// TIA Portal project "Tuan5" (V16)

(* hardware
DEVICE "S7-1200 station_1"  S7-1200 Station
   slot 0: "Rack_0"  S7-1200 Rack  Rack  V1.0
   slot 1: "PLC_1"  CPU 1214C AC/DC/Rly  6ES7 214-1BG40-0XB0  V4.2
*)

// ===== PLC "PLC_1"  CPU 1214C AC/DC/Rly =====

VAR_GLOBAL   // PLC tag table "Default tag table"
   "Stop" AT %I1.2 : Bool;
   "Quay_thuan" AT %Q0.6 : Bool;
   "Quay_nguoc" AT %Q0.7 : Bool;
   "Start" AT %I1.1 : Bool;
   "Tag_5" AT %I0.1 : Bool;
   "Tag_6" AT %M0.0 : Bool;
   "Tag_7" AT %M0.1 : Bool;
   "Time" AT %MD0 : DWord;
   "Tag_8" AT %M0.3 : Bool;
   "Tag_1" AT %M0.2 : Bool;
   "Tag_2" AT %M2.0 : Bool;
   "Tag_3" AT %Q8.1 : Bool;
   "Tag_4" AT %M0.5 : Bool;
   "Tag_9" AT %M0.4 : Bool;
END_VAR

// folder: System blocks/Program resources

DATA_BLOCK "T1"   // DB1
{ S7_Optimized_Access := 'TRUE' }
AUTHOR : Simatic
FAMILY : IEC
NAME : IEC_TMR
VERSION : 1.0
// stored: InstanceOfName IEC_TIMER
"IEC_TIMER"
BEGIN
END_DATA_BLOCK

DATA_BLOCK "T2"   // DB2
{ S7_Optimized_Access := 'TRUE' }
AUTHOR : Simatic
FAMILY : IEC
NAME : IEC_TMR
VERSION : 1.0
// stored: InstanceOfName IEC_TIMER
"IEC_TIMER"
BEGIN
END_DATA_BLOCK

// folder: (top level)

ORGANIZATION_BLOCK "Main"   // OB1, LAD, ProgramCycle
TITLE = "Main Program Sweep (Cycle)"
{ S7_Optimized_Access := 'TRUE' }
VERSION : 0.1
   VAR_INPUT
      Initial_Call : Bool;   // Initial call of this OB
      Remanence : Bool;   // =True, if remanent data are available
   END_VAR
BEGIN

REGION Network 1
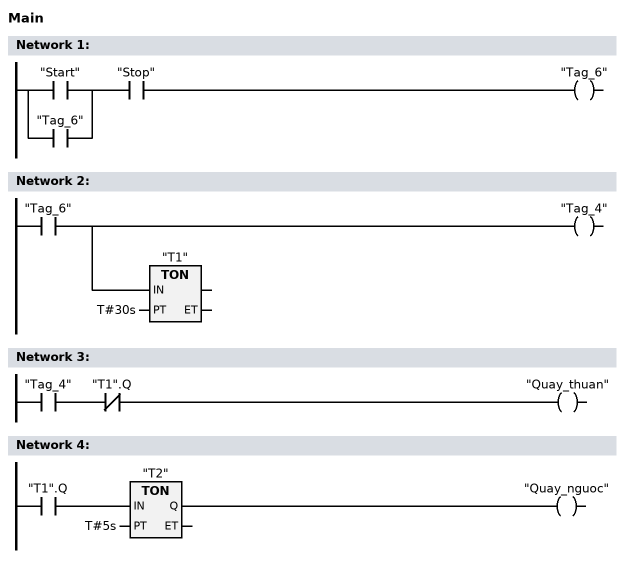
   RUNG wire#powerrail
      Contact( "Start" )
      wire#w1
      Contact( "Stop" )
      Coil( "Tag_6" )
   END_RUNG
   RUNG wire#powerrail
      Contact( "Tag_6" )
   END_RUNG wire#w1
   // the same network as SCL:
   "Tag_6" := ("Start" OR "Tag_6") AND "Stop";
END_REGION

REGION Network 2
   "Tag_4" := "Tag_6";
   "T1".TON(IN := "Tag_6", PT := T#30s);
END_REGION

REGION Network 3
   RUNG wire#powerrail
      Contact( "Tag_4" )
      I_Contact( "T1".Q )
      Coil( "Quay_thuan" )
   END_RUNG
   // the same network as SCL:
   "Quay_thuan" := "Tag_4" AND NOT "T1".Q;
END_REGION

REGION Network 4
   "T2".TON(IN := "T1".Q, PT := T#5s);
   "Quay_nguoc" := "T2".Q;
END_REGION
END_ORGANIZATION_BLOCK